FUNCTION_BLOCK SafetyHydraulicsWidget
VAR_INPUT
END_VAR
VAR_OUTPUT
	actualStatus : StatusWidget;
END_VAR
VAR_IN_OUT
	ref : SafetyHydraulics;
END_VAR
VAR
END_VAR


actualStatus(text  := ref.actualStatus,
             color := HealthBusyToColor(healthStatus := ref.statuses.healthStatus, busyStatus := ref.statuses.busyStatus));

END_FUNCTION_BLOCK

(* stored: Version 1.1.0.1, ProductVersion 3.1.4018.5
   POU SafetyHydraulicsWidget: Id {24a9a5c7-1b79-4fb0-a50a-1c0050de5a46}, SpecialFunc None *)
